{attribute 'GeneratedUsingTerminal: EK1122-0000-0018'}
{attribute addProperty BoxType "EK1122-0000-0018"}
{attribute addProperty Id "Term_17_EK1100Term_17_EK1100_B932616E164"}
{attribute addProperty CRC "3811576148"}
{attribute addProperty Size "164"}
TYPE Term_16_EK1122_E3300954 EXTENDS EK1122_1FC0878B :
STRUCT
	{attribute addProperty Name "Term_17_EK1100"}
	{attribute addProperty PreviousPort "Term 16 (EK1122) : D"}
	Term_17_EK1100 : Term_17_EK1100_B932616E;
END_STRUCT
END_TYPE

(* stored: Version 1.2.0.0, ProductVersion 3.1.4024.9
   DUT Term_16_EK1122_E3300954: Id {c57d63e1-7d34-0c16-357b-ffa6d2eb3802} *)
